FUNCTION TryConvert_SINT_TO_SINT : BOOL
VAR_INPUT
	in : SINT;
	out : REFERENCE TO SINT;
END_VAR

out := in;
TryConvert_SINT_TO_SINT := TRUE;

END_FUNCTION

(* stored: Version 1.1.0.1, ProductVersion 3.1.4024.12
   POU TryConvert_SINT_TO_SINT: Id {c7b9d565-70e8-41eb-98ce-cb3bdba3183d}, SpecialFunc None *)
